Fanuc KAREL source: RMCN_ALERT.kl

PROGRAM T
%NOLOCKGROUP
VAR
 v0 : STRING[40]
 v1 : STRING[40]
 v2 : STRING[40]
 v3 : STRING[40]
 v4 : INTEGER
BEGIN
 RMCN_ALERT(v0, v1, v2, v3, v4)
END T
